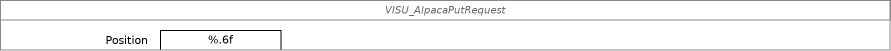
VISUALIZATION VISU_AlpacaPutMove  // 891x51
VAR_IN_OUT
	stInstance : ST_AlpacaPutMove;
END_VAR
    Frame (0,0 891x20)
        shows VISU_AlpacaPutRequest(stInstance := stInstance)
    Label (50,30 101x21), "Position"
    Rectangle (160,30 121x20), "%.6f", text variable: stInstance.i_Position
        OnMouseClick: write the text variable via Default
END_VISUALIZATION

(* stored: Version 1.1.0.1, ProductVersion 3.1.4024.12
   Visu VISU_AlpacaPutMove: Id {b605d9e9-05d4-4f7b-9f1e-ee5da26e06c9} *)
